PROGRAM RunTCP
VAR
	fbTcpServer 	: FB_TcpServer;
	SrvNetId		: STRING := '';
	ServerAddress 	: STRING := '';
	ServerPort 		: UDINT := 24100;
	
	sResponse		: STRING;
	sCommand		: STRING;
	bBusy			: BOOL;
	err				: BOOL;
	errid			: UDINT;
	
	(*
//	blinkLeft : BOOL;
//	blinkRight : BOOL;
//	lightFront : BOOL;
//	lightRear : BOOL;
//	lightBrake : BOOL;

	LightsFront   : BOOL;
	LightsRear 	: BOOL;
	LightsBrake	: BOOL;
	LightsReverse : BOOL;
    BlinkerLeft     : BOOL;
    BlinkerRight    : BOOL;*)
	
END_VAR

fbTcpServer(
	NetId:= SrvNetId, 
	ServerAdr:= ServerAddress, 
	ServerPort:= ServerPort, 
	sSend := sResponse,
	sReceive=> sCommand, 
	bBusy=> bBusy, 
	err=> err, 
	errid=> errid);
	
	sResponse := sCommand;
	
	TCPTimeOut();
	Lights();
	FnR_Switch();
	SafetyMode();
	GetSpeedSteer();

END_PROGRAM

(* stored: Version 1.1.0.1, ProductVersion 3.1.4024.3
   POU RunTCP: Id {807811c6-709a-444f-a511-9b1280f909c8}, SpecialFunc None *)
